// Mitsubishi GX Works2 project: backup code   PLC: FX1N/FX1NC

// global labels: Global1
VAR_GLOBAL
  ONOFF AT M0 : BOOL;
  Lock AT M1 : BOOL;
  Inducprox AT X000 : BOOL;
  PIR AT X001 : BOOL;
  LED AT Y000 : BOOL;
  Buzzer AT Y001 : BOOL;
  Motor1 AT Y002 : BOOL;  (* สามารถตั้งค่าความเร็ว และเวลาที่หมุนได้ *)
  Indhold AT M2 : BOOL;
  PIRhold AT M3 : BOOL;
  Motor2 AT Y003 : BOOL;  (* ขึ้นกับความกว้างที่ต้องการเปิดประตู *)
  Sound AT M4 : BOOL;
  Motor1hold AT M6 : BOOL;
  Motot2hold AT M7 : BOOL;
END_VAR

PROGRAM MAIN
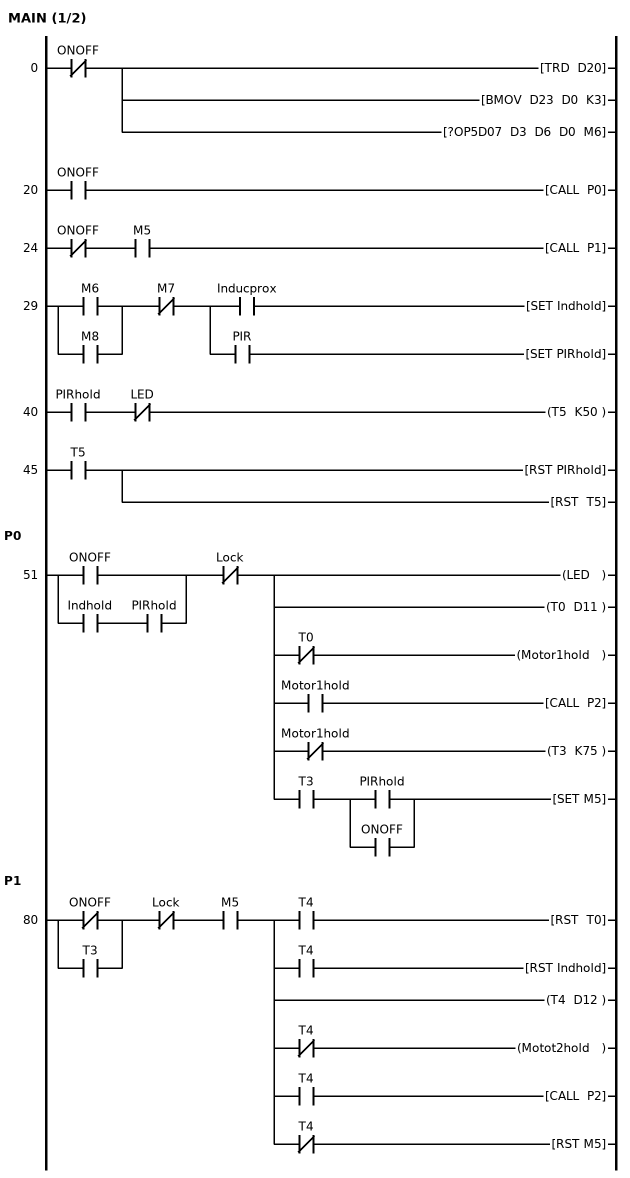
0     LDI     ONOFF
      TRD     D20
      BMOV    D23 D0 K3
      ?OP5D07 D3 D6 D0 M6
20    LD      ONOFF
      CALL    P0
24    LDI     ONOFF
      AND     M5
      CALL    P1
29    LD      M6
      OR      M8
      ANI     M7
      MPS
      AND     Inducprox
      SET     Indhold
      MPP
      AND     PIR
      SET     PIRhold
40    LD      PIRhold
      ANI     LED
      OUT     T5 K50
45    LD      T5
      RST     PIRhold
      RST     T5
      P0
51    LD      ONOFF
      LD      Indhold
      AND     PIRhold
      ORB
      ANI     Lock
      OUT     LED
      OUT     T0 D11
      MPS
      ANI     T0
      OUT     Motor1hold
      MRD
      AND     Motor1hold
      CALL    P2
      MRD
      ANI     Motor1hold
      OUT     T3 K75
      MPP
      AND     T3
      LD      PIRhold
      OR      ONOFF
      ANB
      SET     M5
      P1
80    LDI     ONOFF
      OR      T3
      ANI     Lock
      AND     M5
      MPS
      AND     T4
      RST     T0
      MRD
      AND     T4
      RST     Indhold
      MPP
      OUT     T4 D12
      MPS
      ANI     T4
      OUT     Motot2hold
      MRD
      AND     T4
      CALL    P2
      MPP
      ANI     T4
      RST     M5
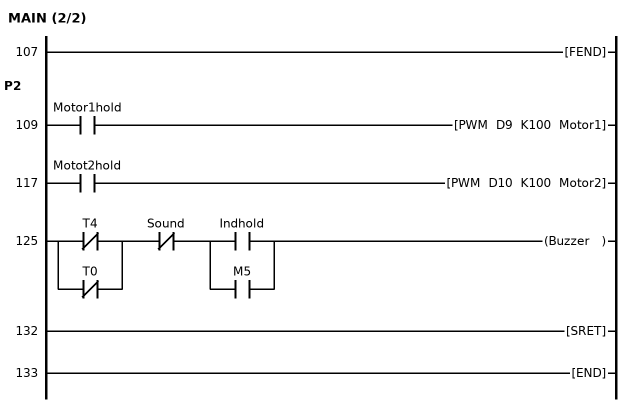
107   FEND
      P2
109   LD      Motor1hold
      PWM     D9 K100 Motor1
117   LD      Motot2hold
      PWM     D10 K100 Motor2
125   LDI     T4
      ORI     T0
      ANI     Sound
      LD      Indhold
      OR      M5
      ANB
      OUT     Buzzer
132   SRET
133   END
END_PROGRAM
